(* Schneider Machine Expert - Basic project p7, file version 1.8.0.0 *)
(* ProjectInformations: Name=New project *)

HARDWARE
  Cpu 0: TM221CE16R
  EthernetConfiguration: NetworkName=M221, IpAllocationMode=FixedAddress, IpAddress=192.168.162.202, SubnetMask=255.255.255.0
  SerialLineConfiguration: Baud=Baud19200, Parity=ParityEven, DataBits=DataBits8, StopBits=StopBits1, PhysicalMedium=PhysicalMediumRs485, TransmissionMode=TransmissionModeModbusRtu, SlaveId=1, Addressing=SlaveAddressing
  MastTask: UsePeriodScanMode=false, PeriodScan=100
  FastTask: Period=255
  CpuBehavior: StartingMode=StartAsPreviousState, AutoSaveRamOnEeprom=true, WatchdogPeriod=250

SYMBOLS  (address, symbol, comment, settings)
  %S6       SB_TB1S  "Time base of 1 s generated by an internal clock"

POU New POU
  (* SectionNumber=1 *)

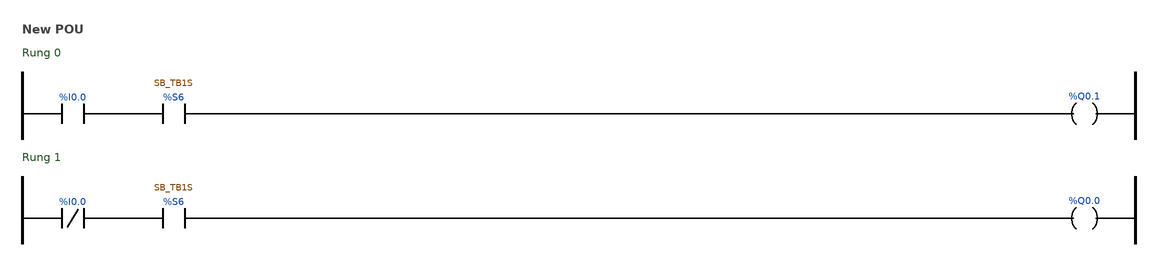

// Rung 0
  LD %I0.0
  AND %S6                 (* SB_TB1S *)
  ST %Q0.1
  // as ST:
  //   %Q0.1 := %I0.0 AND SB_TB1S;

// Rung 1
  LDN %I0.0
  AND %S6                 (* SB_TB1S *)
  ST %Q0.0
  // as ST:
  //   %Q0.0 := NOT %I0.0 AND SB_TB1S;
